Yaskawa INFORM job: MASTER_SCIANA_R1_MOD.JBI

/JOB
//NAME MASTER_SCIANA_R1_MOD
///FOLDERNAME SCIANA_WYPYCHAJACA_V19B_V20
//POS
///NPOS 54,54,54,0,0,0
///TOOL 0
///POSTYPE PULSE
///PULSE
C00000=5011,38780,33406,-3752,88219,85582
C00001=5011,38780,33406,-3752,88219,85582
C00002=5012,38778,33409,-3767,88218,85582
C00003=5011,38780,33406,-3752,88219,85582
C00004=-13644,-92138,-120638,38655,87204,86250
C00005=-13644,-92138,-120638,38655,87204,86250
C00006=-3569,-152063,-129797,3896,35885,81269
C00007=13512,109275,27441,-16100,94054,76800
C00008=-97801,-92951,-68020,-42573,91743,12282
C00009=26932,41391,-30369,6536,105272,62664
C00010=147750,-31965,-71698,11557,98758,54427
C00011=28105,107103,24913,-6745,88279,69024
C00012=1503,48046,-28403,-12258,96069,81953
C00013=-64345,6993,-34056,-5678,86941,71323
C00014=-88506,-94181,-91931,-694,81235,59832
C00015=-88506,-94181,-91931,-709,81235,59832
C00016=-46304,-10837,-44678,-4666,86111,69253
C00017=29020,137920,39663,-11730,94813,86069
C00018=29020,137920,39663,-11730,94813,86069
C00019=-78395,-65747,-78398,-11730,94813,86069
C00020=112867,-145355,-130280,-83721,-18285,-930
C00021=112867,-145355,-130280,5739,-2626,-930
C00022=46432,-159370,-130280,2544,61420,-930
C00023=19143,-90916,-90036,-16768,72453,41097
C00024=13148,3851,-75147,6736,62300,60674
C00025=15005,124146,46234,-8348,94498,60234
C00026=22665,120049,18248,-11675,101032,82300
C00027=3857,107043,326,1084,102018,80372
C00028=3857,107043,326,1084,102018,80372
C00029=20488,129728,35048,-15297,94679,79335
C00030=23133,116740,10365,-10832,101628,84944
C00031=23133,116740,10365,-10832,101628,84944
C00032=-99911,-177915,-134930,14535,-6478,4116
C00033=-114272,-169051,-129428,11712,720,2256
C00034=-10051,-169051,-129428,11712,75776,2256
C00035=2132,-35541,-62189,-16099,8927,75121
C00036=9572,-20991,-102984,-16549,97127,59885
C00037=-1999,180198,107788,-13936,86373,83899
C00038=4050,-131452,-116592,-2442,-516,-21528
C00039=32544,80755,19414,-44490,116423,65030
C00040=3198,-156648,-132716,2511,-14356,-31810
C00041=-16374,-140825,-127462,-11617,89672,81747
C00042=119308,-140825,-127462,-11617,12243,81747
C00043=119308,-140825,-127462,-11617,12243,81747
C00044=175566,-140825,-127462,-11617,41655,77429
C00045=142654,-146608,-121681,-23127,-3079,28805
C00046=21373,-146309,-121603,-17654,-2866,26368
C00047=5748,-150278,-123121,-19822,31163,-82107
C00048=5748,-150278,-123121,-19822,31163,-82107
C00049=6111,-145918,-120649,-19707,32112,-79579
C00050=-21526,-164536,-89902,40074,64113,11441
C00051=5210,21378,-27343,16666,83947,-8287
C00052=5011,38780,33406,-3752,88219,85582
C00053=5011,38780,33406,-3752,88219,85582
BC00000=61339,583433,800287
BC00001=61339,583433,1035649
BC00002=61340,583436,1035643
BC00003=61339,583433,1035649
BC00004=194821,433358,1073901
BC00005=194821,473945,1073901
BC00006=85972,554727,1026528
BC00007=106484,483988,1039881
BC00008=365145,1359,801155
BC00009=165105,11813,1033268
BC00010=337965,17193,1016408
BC00011=87809,401940,1060967
BC00012=177539,404256,1041609
BC00013=271646,226929,981220
BC00014=294910,15771,909310
BC00015=294911,15771,909309
BC00016=304749,174467,1044799
BC00017=86869,457719,1075157
BC00018=86869,457719,1075157
BC00019=315222,408143,1075157
BC00020=393418,389878,1050203
BC00021=393418,5524,1050203
BC00022=393418,5524,1050203
BC00023=344649,733,1067002
BC00024=4442,404413,1013854
BC00025=109002,65001,1068359
BC00026=138740,5300,1068817
BC00027=125260,23786,1075157
BC00028=125260,23786,1075157
BC00029=137052,525583,1075158
BC00030=125260,578,1075157
BC00031=125260,578,1075157
BC00032=18154,534183,651605
BC00033=4712,11801,676331
BC00034=4712,11801,676331
BC00035=13234,23982,1061417
BC00036=12870,140,1075170
BC00037=82357,456758,1075208
BC00038=21826,498643,1037907
BC00039=34258,544306,720525
BC00040=24328,497765,1075175
BC00041=106517,503923,1075158
BC00042=254539,503923,1075158
BC00043=385321,205052,1075158
BC00044=385321,140478,1075158
BC00045=398173,254870,1075173
BC00046=236760,481426,1075173
BC00047=208302,536639,1074746
BC00048=208302,536639,1074746
BC00049=206156,6818,1073429
BC00050=121998,847,1075175
BC00051=124816,585235,1074582
BC00052=61339,583433,1035649
BC00053=61339,583433,800287
EC00000=0,1
EC00001=0,1
EC00002=830412,556476
EC00003=0,1
EC00004=-798147,556474
EC00005=-798147,556474
EC00006=-1,0
EC00007=0,0
EC00008=0,0
EC00009=-1,0
EC00010=-1,0
EC00011=-1,0
EC00012=-1,0
EC00013=-1,0
EC00014=-1,0
EC00015=-368461,-562332
EC00016=-234121,-277023
EC00017=-1,0
EC00018=-1,0
EC00019=-1,0
EC00020=798157,0
EC00021=798157,0
EC00022=798157,0
EC00023=798156,0
EC00024=798157,-556476
EC00025=-620788,-556475
EC00026=-399079,-556476
EC00027=0,-556476
EC00028=0,-556476
EC00029=0,0
EC00030=798157,556476
EC00031=798157,556476
EC00032=798157,1112952
EC00033=798157,1112952
EC00034=798157,1112952
EC00035=798150,1112953
EC00036=798150,1112953
EC00037=709473,1112952
EC00038=1596314,554480
EC00039=1596314,556476
EC00040=1596314,0
EC00041=1596314,0
EC00042=1596314,0
EC00043=1596314,0
EC00044=1596314,0
EC00045=1596314,0
EC00046=1596314,0
EC00047=1596314,1112952
EC00048=1596314,1112952
EC00049=1152894,-556476
EC00050=1218674,-556476
EC00051=923702,561565
EC00052=0,1
EC00053=0,1
//INST
///DATE 2025/04/30 17:22
///ATTR SC,RW
///GROUP1 RB1,BS1
///GROUP2 ST1
NOP
MOVJ C00000 BC00000 VJ=100.00  +MOVJ EC00000 VJ=100.00
MOVJ C00001 BC00001 VJ=100.00  +MOVJ EC00001 VJ=100.00
COMM MOVJ C00002 BC00002 VJ=100.00  +MOVJ EC00002 VJ=100.00
COMM PAUSE
PAUSE
COMM 'UWAGA!!!!
COMM 'SCIAGNAC UCHWYTY SCIANY
MOVJ C00003 BC00003 VJ=100.00  +MOVJ EC00003 VJ=100.00
COMM DOUT OT#(1433) ON
DOUT OT#(1434) ON
CALL JOB:0_-90
CALL JOB:R1_W01(KAMERA)(0,-90)
CALL JOB:125_90
CALL JOB:R1_W12(125,90)(KAMERA)
CALL JOB:-90_90
CALL JOB:R1_W26(-90,90)(KAMERA)
COMM CALL JOB:R1_W26(-90,90)(KAMERA)
CALL JOB:R1_W23(-90,90)(KAMERA)KM-OK
MOVJ C00004 BC00004 VJ=100.00  +MOVJ EC00004 VJ=40.00
CALL JOB:R1_W24(-90,90)KM-OK
MOVJ C00005 BC00005 VJ=100.00  +MOVJ EC00005 VJ=100.00
MOVJ C00006 BC00006 VJ=100.00  +MOVJ EC00006 VJ=100.00
'KONIEC SPAWANIA ZE SLEDZENIEM
'KAMERA SERVO ROBOT
'----------------------
CALL JOB:ONLYCUT-R1_LONG
CALL JOB:0_0
MOVJ C00007 BC00007 VJ=100.00  +MOVJ EC00007 VJ=30.00
MOVJ C00008 BC00008 VJ=100.00  +MOVJ EC00008 VJ=40.00
CALL JOB:R1_W03,5,7(0,0)OK-KM
CALL JOB:ONLYCUT-R1_LONG
MOVJ C00009 BC00009 VJ=100.00  +MOVJ EC00009 VJ=40.00
MOVJ C00010 BC00010 VJ=100.00  +MOVJ EC00010 VJ=40.00
CALL JOB:R1_W02,4,6(0_0)_KM-OK
MOVJ C00011 BC00011 VJ=100.00  +MOVJ EC00011 VJ=100.00
CALL JOB:CLEAN-R1_LONG
CALL JOB:R1_W14,16(0,0)OK-KM
CALL JOB:CLEAN-R1_LONG
CALL JOB:R1_W13,15(0,0)KM-OK
CALL JOB:ONLYCUT-R1_LONG
MOVJ C00012 BC00012 VJ=100.00  +MOVJ EC00012 VJ=100.00
MOVJ C00013 BC00013 VJ=100.00  +MOVJ EC00013 VJ=100.00
MOVJ C00014 BC00014 VJ=100.00  +MOVJ EC00014 VJ=100.00
MOVJ C00015 BC00015 VJ=50.00  +MOVJ EC00015 VJ=50.00
CALL JOB:R1_W17,20,22(0,0)OK-KMNEW
MOVJ C00016 BC00016 VJ=40.00  +MOVJ EC00016 VJ=40.00
MOVJ C00017 BC00017 VJ=40.00  +MOVJ EC00017 VJ=25.00
CALL JOB:CLEAN-R1_LONG
MOVJ C00018 BC00018 VJ=40.00  +MOVJ EC00018 VJ=40.00
MOVJ C00019 BC00019 VJ=40.00  +MOVJ EC00019 VJ=40.00
'DODANE SEARCH
CALL JOB:R1_W18,19,21(0,0)_KM-OKNEW_MP
COMM CALL JOB:R1_W18,19,21(0,0)_KM-OKNEW
CALL JOB:CLEAN-R1_LONG
CALL JOB:R1_W30(0,0)OK-KM
CALL JOB:ONLYCUT-R1_LONG
CALL JOB:R1_W33(0,0)KM-OK
CALL JOB:CLEAN-R1_LONG
CALL JOB:R1_W31(0,0)_KM-OK
'----------------------
'SPAWANIE DLA POZYCJI 90_0
CALL JOB:90_0
MOVJ C00020 BC00020 VJ=100.00  +MOVJ EC00020 VJ=100.00
MOVJ C00021 BC00021 VJ=100.00  +MOVJ EC00021 VJ=100.00
MOVJ C00022 BC00022 VJ=100.00  +MOVJ EC00022 VJ=100.00
MOVJ C00023 BC00023 VJ=100.00  +MOVJ EC00023 VJ=40.00
CALL JOB:CLEAN-R1_LONG
CALL JOB:R1_W27-A3(90,0)OK-KM
CALL JOB:ONLYCUT-R1_LONG
CALL JOB:R1_W27-A5(90,0)OK-KM_MOD
CALL JOB:CLEAN-R1_LONG
CALL JOB:R1_W35-36-A2(90,0)KM-OK_MOD
CALL JOB:ONLYCUT-R1_LONG
CALL JOB:R1_W45-48(90,0)KM-OK
'W39-53
CALL JOB:R1_W39(90,0)R2
'---------------------
'SPAWANIE DLA POZYCJI 90_-90
CALL JOB:90_-90
MOVJ C00024 BC00024 VJ=100.00  +MOVJ EC00024 VJ=100.00
CALL JOB:CLEAN-R1_LONG
CALL JOB:R1_W27-A2(90,-90)POPR-KM-OK_MOD
CALL JOB:ONLYCUT-R1_LONG
COMM CALL JOB:R1_W29-KM-NOWY
'POPRAWA SEARCH
CALL JOB:R1_W29-KM-NOWY-MP
'---------------------
'ZMIANA POZYCJI SPAWANIA -70_-90
'AWOK
CALL JOB:-70_-90
MOVJ C00025 BC00025 VJ=100.00  +MOVJ EC00025 VJ=40.00
CALL JOB:CLEAN-R1_LONG
CALL JOB:R1_W09,10(-70,-90)
CALL JOB:ONLYCUT-R1_LONG
CALL JOB:R1_W08,11(-70,-90)_KM-OK
CALL JOB:ONLYCUT-R1_LONG
CALL JOB:R1_W66-67(-70,-90)KM-OK
CALL JOB:CLEAN-R1_LONG
CALL JOB:R1_W66-W67(-70,-90)KM-OK
'---------------------
'AWOK
'ZMIANA POZYCJI SPAWANIA -90_-90
CALL JOB:-90_-90
CALL JOB:ONLYCUT-R1_LONG
CALL JOB:R1_W68-69(-90,-90)KM-OK
CALL JOB:CLEAN-R1_LONG
CALL JOB:R1_W68-69(-90,-90)KM-OK-R2
CALL JOB:ONLYCUT-R1_LONG
CALL JOB:R1_W70(-90,-90)KM-OK
MOVJ C00026 BC00026 VJ=100.00  +MOVJ EC00026 VJ=100.00
'ZMIANA POZYCJI SPAWANIA -45_-90
CALL JOB:-45_-90
CALL JOB:CLEAN-R1_LONG
CALL JOB:R1_W72(-45,-90)KM-OK
CALL JOB:CLEAN-R1_LONG
CALL JOB:R1_W72(-45,-90)R2
MOVJ C00027 BC00027 VJ=100.00  +MOVJ EC00027 VJ=100.00
'ZMIANA POZYCJI SPAWANIA 0_-90
CALL JOB:0_-90
MOVJ C00028 BC00028 VJ=100.00  +MOVJ EC00028 VJ=30.00
CALL JOB:ONLYCUT-R1_LONG
CALL JOB:R1_W73(0,-90)KM-OK
'ZMIANA POZYCJI SPAWANIA 0_0
'AWOK
MOVJ C00029 BC00029 VJ=100.00  +MOVJ EC00029 VJ=100.00
CALL JOB:ONLYCUT-R1_LONG
CALL JOB:R1_72,2(0,0)KM-OK_MOD
CALL JOB:ONLYCUT-R1_LONG
CALL JOB:R1_72,2(0,0)R2_MOD
'ZMIANA POZYCJI SPAWANIA 80_0
CALL JOB:80_0
CALL JOB:CLEAN-R1_LONG
CALL JOB:R1_W43-44-A1(80,0))KM-OK_MOD
'ZMIANA POZYCJI SPAWANIA 90_90
MOVJ C00030 BC00030 VJ=100.00  +MOVJ EC00030 VJ=30.00
CALL JOB:CLEAN-R1_LONG
MOVJ C00031 BC00031 VJ=100.00  +MOVJ EC00031 VJ=15.00
CALL JOB:R1_W49-52-A2(90,90)KM-OK
CALL JOB:ONLYCUT-R1_LONG
CALL JOB:R1_W53-A2(90,90)
'ZMIANA POZYCJI SPAWANIA 90_180
CALL JOB:90_180
CALL JOB:CLEAN-R1_LONG
MOVJ C00032 BC00032 VJ=100.00  +MOVJ EC00032 VJ=100.00
MOVJ C00033 BC00033 VJ=100.00  +MOVJ EC00033 VJ=100.00
MOVJ C00034 BC00034 VJ=100.00  +MOVJ EC00034 VJ=100.00
CALL JOB:R1_W27-A4(90,180)KM-OK_MOD
SFTOF
MOVJ C00035 BC00035 VJ=100.00  +MOVJ EC00035 VJ=100.00
CALL JOB:ONLYCUT-R1_LONG
CALL JOB:R1_W35-36-A1(90,180)KM-OK_MOD
MOVJ C00036 BC00036 VJ=100.00  +MOVJ EC00036 VJ=10.00
'SPR PRZEJAZDY
CALL JOB:CLEAN-R1_LONG
CALL JOB:R1_W49-52-A1(90,180)KM-OK
CALL JOB:ONLYCUT-R1_LONG
CALL JOB:R1_W27-A4(90,180)_KM_OKR2
CALL JOB:ONLYCUT-R1_LONG
CALL JOB:R1_W53-A1(90,180)R2
'ZMIANA POZYCJI SPAWANIA 80_180
CALL JOB:80_180
CALL JOB:CLEAN-R1_LONG
MOVJ C00037 BC00037 VJ=40.00  +MOVJ EC00037 VJ=40.00
CALL JOB:R1_W43-44-A2(80,180)KM-OK_MOD
'ZMIANA POZYCJI SPAWANIA 180_0
CALL JOB:180_90
MOVJ C00038 BC00038 VJ=100.00  +MOVJ EC00038 VJ=40.00
CALL JOB:ONLYCUT-R1_LONG
CALL JOB:R1_W43-44-A3(0,180)_MOD
MOVJ C00039 BC00039 VJ=100.00  +MOVJ EC00039 VJ=40.00
CALL JOB:180_0
MOVJ C00040 BC00040 VJ=100.00  +MOVJ EC00040 VJ=40.00
CALL JOB:ONLYCUT-R1_LONG
MOVJ C00041 BC00041 VJ=100.00  +MOVJ EC00041 VJ=100.00
MOVJ C00042 BC00042 VJ=100.00  +MOVJ EC00042 VJ=100.00
MOVJ C00043 BC00043 VJ=100.00  +MOVJ EC00043 VJ=100.00
MOVJ C00044 BC00044 VJ=100.00  +MOVJ EC00044 VJ=100.00
CALL JOB:R1_W49-52-A5(180,0)KM-OK
MOVJ C00045 BC00045 VJ=100.00  +MOVJ EC00045 VJ=20.00
MOVJ C00046 BC00046 VJ=100.00  +MOVJ EC00046 VJ=100.00
CALL JOB:CLEAN-R1_LONG
CALL JOB:R1_W53-A5(180,0)KM-OK_R2
'ZMIANA POZYCJI SPAWANIA 180_180
MOVJ C00047 BC00047 VJ=100.00  +MOVJ EC00047 VJ=100.00
CALL JOB:CLEAN-R1_LONG
MOVJ C00048 BC00048 VJ=40.00  +MOVJ EC00048 VJ=100.00
'ZMIANA POZYCJI SPAWANIA 130_-90
CALL JOB:130_-90
MOVJ C00049 BC00049 VJ=100.00  +MOVJ EC00049 VJ=100.00
CALL JOB:R1_W63-A2(130,-90)(JEDENR)KM-OK
'ZMIANA POZYCJI SPAWANIA 120_-90
CALL JOB:120_-90
MOVL C00050 BC00050 V=1000.0  +MOVJ EC00050 VJ=100.00
CALL JOB:CLEAN-R1_LONG
CALL JOB:R1_W63-A1(120,-90)KM-OK
CALL JOB:CLEAN-R1_LONG
CALL JOB:R1_W63-A1(120,-90)KM-OK_R2
COMM DOUT OT#(1433) OFF
DOUT OT#(1434) OFF
COMM MOVJ C00051 BC00051 VJ=100.00  +MOVJ EC00051 VJ=100.00
COMM PAUSE
COMM 'UWAGA!!!!
COMM 'ZALOZ UCHYWTY DO SCIANY
CALL JOB:0_0
MOVJ C00052 BC00052 VJ=100.00  +MOVJ EC00052 VJ=0.78
MOVJ C00053 BC00053 VJ=100.00  +MOVJ EC00053 VJ=100.00
PAUSE
SFTOF
END
